Universal Robots PolyScope program: program 2.urp

Program program 2 (installation=default directory=/ursim/programs createdIn=3.15.8.106339 lastSavedIn=3.15.8.106339 robotSerialNumber=2018359999)
Calibrated DH parameters: a=[0, -0.425, -0.39225, 0, 0, 0]; d=[0.089159, 0, 0, 0.10915, 0.09465, 0.0823]; alpha=[1.570796, 0, 0, 1.570796, -1.570796, 0]; deltaTheta=[0, 0, 0, 0, 0, 0]
Robot Program (runOnlyOnce=false)
  Set DigitalOutput pin=digital_out[0]; digitalValue=1
  Wait Sleep waitTime=0.01
  Popup Message (haltProgram=false message=El control será compartido con un controlador externo (ROS2) presiona OK para continuar :) inputType=Text)
  Wait Sleep waitTime=5
  Script: textmsg("esperando el control externo desde ROS2")
  URCap External Control (External Control, FZI Research Center for Information Technology)
